// TIA Portal project "FBMECaSYSTEM_COUNTER" (V17)

(* hardware
DEVICE "HMI_1"  KTP900 Basic PN
   slot 0: "HMI_1"  KTP900 Basic PN  6AV2 123-2JB03-0AX0  17.0.0.0
   slot 1: "HMI_RT_1"  KTP900 Basic PN  6AV2 123-2JB03-0AX0  17.0.0.0
   slot 5: "HMI_1.IE_CP_1"  PROFINET Interface  17.0.0.0
      slot 1: "PROFINET Interface_1"  PROFINET Interface
         slot 1: "Port_1"  Port
DEVICE "S7-1200 station_1"  S7-1200 Station
   slot 0: "Rack_0"  S7-1200 Rack  Rack  V1.0
   slot 1: "PLC_1"  CPU 1214C AC/DC/Rly  6ES7 214-1BG40-0XB0  V4.5
*)

// ===== PLC "PLC_1"  CPU 1214C AC/DC/Rly =====

VAR_GLOBAL   // PLC tag table "Default tag table"
   "NbPersonneEntree" AT %IW10 : Int;
   "NbPersonneSortie" AT %IW14 : Int;
   "EntrerValider" AT %I20.0 : Bool;
   "SortieValider" AT %I20.1 : Bool;
   "FrontEntrerValider" AT %I20.2 : Bool;
   "FrontSortieValider" AT %I20.3 : Bool;
   "NbPersonnneInSide" AT %IW12 : Int;
   "NbPersonneTotalAutorise" AT %IW16 : Int;
   "NbPeronneRestant" AT %IW18 : Int;
   "EntreePMRValider" AT %I20.4 : Bool;
   "SortiePMRValider" AT %I20.5 : Bool;
   "NbPMR" AT %IW22 : Int;
   "FontPMRENtree" AT %I20.6 : Bool;
   "FrontPMRSortie" AT %I20.7 : Bool;
   "SitePleinQuatreVingtPC" AT %I21.0 : Bool;
   "SitePleinCentPC" AT %I21.1 : Bool;
   "FOIS80" AT %IW24 : Int;
   "DIVISER100" AT %IW26 : Int;
   "EtatRempliSite" AT %IW28 : Int;
   "Tag_1" AT %I21.2 : Bool;
   "Tag_2" AT %I21.3 : Bool;
   "Tag_3" AT %I21.4 : Bool;
   "Tag_4" AT %I21.5 : Bool;
END_VAR

ORGANIZATION_BLOCK "Main"   // OB1, LAD, ProgramCycle
TITLE = "Main Program Sweep (Cycle)"
{ S7_Optimized_Access := 'TRUE' }
VERSION : 0.1
   VAR_INPUT
      Initial_Call : Bool;   // Initial call of this OB
      Remanence : Bool;   // =True, if remanent data are available
   END_VAR
   VAR_TEMP   // added for the SCL form of the ladder/FBD networks
      _w1 : Bool;
      _w2 : Bool;
   END_VAR
BEGIN

REGION Network 1: Personne untaire entree
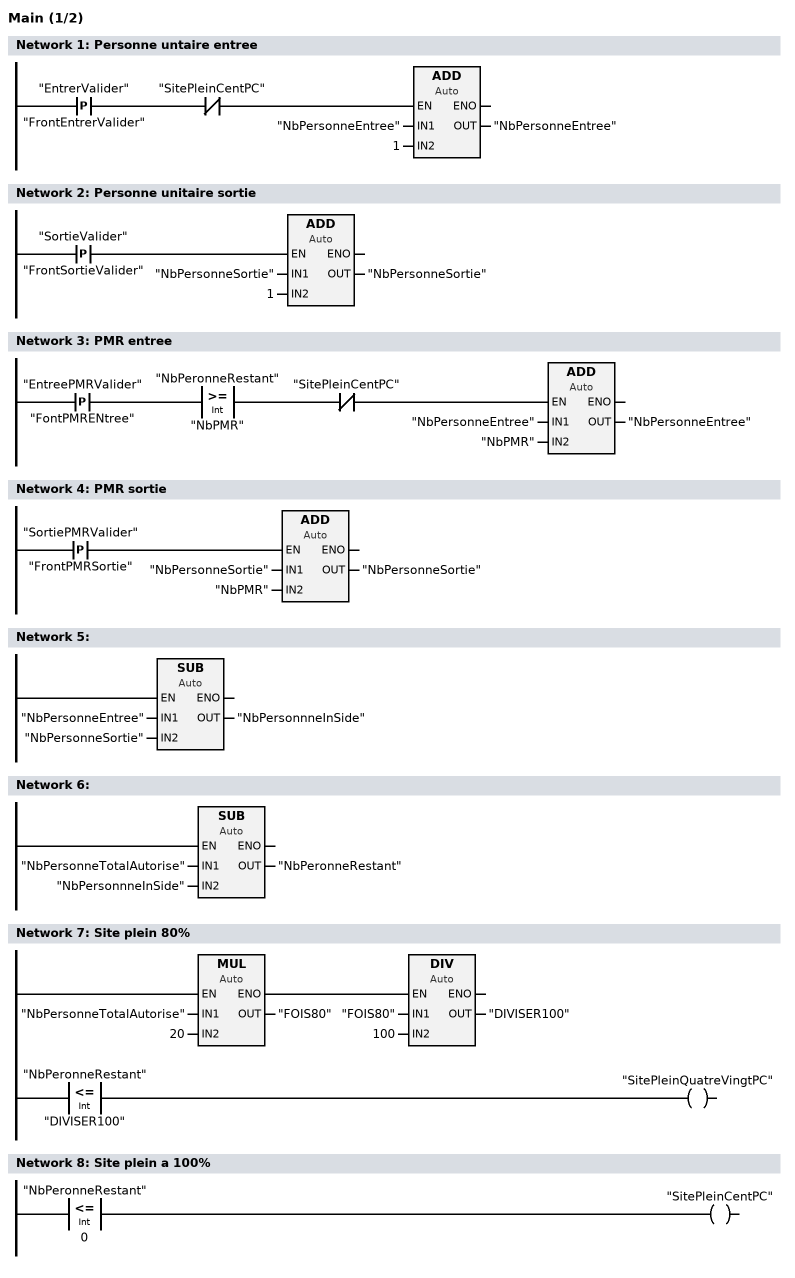
   RUNG wire#powerrail
      P_Contact(operand := "EntrerValider", bit := "FrontEntrerValider")
      I_Contact( "SitePleinCentPC" )
      Add(in1 := "NbPersonneEntree", in2 := 1, out => "NbPersonneEntree")
   END_RUNG
   // the same network as SCL:
   #_w1 := "EntrerValider" AND NOT "FrontEntrerValider";   // rising edge of "EntrerValider"
   "FrontEntrerValider" := "EntrerValider";
   IF #_w1 AND NOT "SitePleinCentPC" THEN "NbPersonneEntree" := "NbPersonneEntree" + 1; END_IF;
END_REGION

REGION Network 2: Personne unitaire sortie
   RUNG wire#powerrail
      P_Contact(operand := "SortieValider", bit := "FrontSortieValider")
      Add(in1 := "NbPersonneSortie", in2 := 1, out => "NbPersonneSortie")
   END_RUNG
   // the same network as SCL:
   #_w1 := "SortieValider" AND NOT "FrontSortieValider";   // rising edge of "SortieValider"
   "FrontSortieValider" := "SortieValider";
   IF #_w1 THEN "NbPersonneSortie" := "NbPersonneSortie" + 1; END_IF;
END_REGION

REGION Network 3: PMR entree
   RUNG wire#powerrail
      P_Contact(operand := "EntreePMRValider", bit := "FontPMRENtree")
      { S7_Templates := "SrcType := Int" } GE_Contact(in1 := "NbPeronneRestant", in2 := "NbPMR")
      I_Contact( "SitePleinCentPC" )
      Add(in1 := "NbPersonneEntree", in2 := "NbPMR", out => "NbPersonneEntree")
   END_RUNG
   // the same network as SCL:
   #_w1 := "EntreePMRValider" AND NOT "FontPMRENtree";   // rising edge of "EntreePMRValider"
   "FontPMRENtree" := "EntreePMRValider";
   IF #_w1 AND ("NbPeronneRestant" >= "NbPMR") AND NOT "SitePleinCentPC" THEN
       "NbPersonneEntree" := "NbPersonneEntree" + "NbPMR";
   END_IF;
END_REGION

REGION Network 4: PMR sortie
   RUNG wire#powerrail
      P_Contact(operand := "SortiePMRValider", bit := "FrontPMRSortie")
      Add(in1 := "NbPersonneSortie", in2 := "NbPMR", out => "NbPersonneSortie")
   END_RUNG
   // the same network as SCL:
   #_w1 := "SortiePMRValider" AND NOT "FrontPMRSortie";   // rising edge of "SortiePMRValider"
   "FrontPMRSortie" := "SortiePMRValider";
   IF #_w1 THEN "NbPersonneSortie" := "NbPersonneSortie" + "NbPMR"; END_IF;
END_REGION

REGION Network 5
   RUNG wire#powerrail
      Sub(in1 := "NbPersonneEntree", in2 := "NbPersonneSortie", out => "NbPersonnneInSide")
   END_RUNG
   // the same network as SCL:
   "NbPersonnneInSide" := "NbPersonneEntree" - "NbPersonneSortie";
END_REGION

REGION Network 6
   RUNG wire#powerrail
      Sub(in1 := "NbPersonneTotalAutorise", in2 := "NbPersonnneInSide", out => "NbPeronneRestant")
   END_RUNG
   // the same network as SCL:
   "NbPeronneRestant" := "NbPersonneTotalAutorise" - "NbPersonnneInSide";
END_REGION

REGION Network 7: Site plein 80%
   RUNG wire#powerrail
      Mul(in1 := "NbPersonneTotalAutorise", in2 := 20, out => "FOIS80")
      Div(in1 := "FOIS80", in2 := 100, out => "DIVISER100")
   END_RUNG
   RUNG wire#powerrail
      { S7_Templates := "SrcType := Int" } LE_Contact(in1 := "NbPeronneRestant", in2 := "DIVISER100")
      Coil( "SitePleinQuatreVingtPC" )
   END_RUNG
   // the same network as SCL:
   "FOIS80" := "NbPersonneTotalAutorise" * 20;
   "DIVISER100" := "FOIS80" / 100;
   "SitePleinQuatreVingtPC" := "NbPeronneRestant" <= "DIVISER100";
END_REGION

REGION Network 8: Site plein a 100%
   RUNG wire#powerrail
      { S7_Templates := "SrcType := Int" } LE_Contact(in1 := "NbPeronneRestant", in2 := 0)
      Coil( "SitePleinCentPC" )
   END_RUNG
   // the same network as SCL:
   "SitePleinCentPC" := "NbPeronneRestant" <= 0;
END_REGION

REGION Network 9
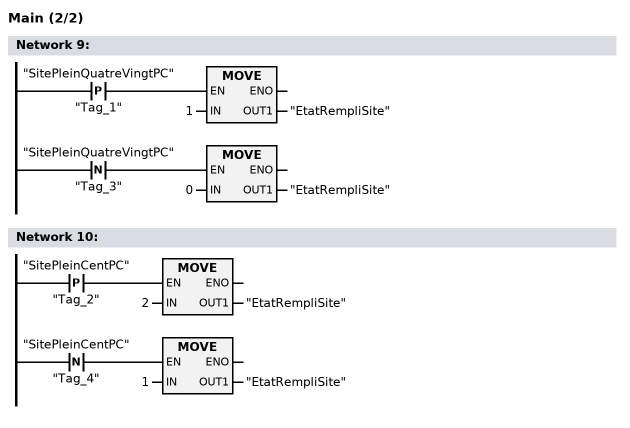
   RUNG wire#powerrail
      P_Contact(operand := "SitePleinQuatreVingtPC", bit := "Tag_1")
      Move(in := 1, out1 => "EtatRempliSite")
   END_RUNG
   RUNG wire#powerrail
      N_Contact(operand := "SitePleinQuatreVingtPC", bit := "Tag_3")
      Move(in := 0, out1 => "EtatRempliSite")
   END_RUNG
   // the same network as SCL:
   #_w1 := "SitePleinQuatreVingtPC" AND NOT "Tag_1";   // rising edge of "SitePleinQuatreVingtPC"
   "Tag_1" := "SitePleinQuatreVingtPC";
   IF #_w1 THEN "EtatRempliSite" := 1; END_IF;
   #_w2 := NOT "SitePleinQuatreVingtPC" AND "Tag_3";   // falling edge of "SitePleinQuatreVingtPC"
   "Tag_3" := "SitePleinQuatreVingtPC";
   IF #_w2 THEN "EtatRempliSite" := 0; END_IF;
END_REGION

REGION Network 10
   RUNG wire#powerrail
      P_Contact(operand := "SitePleinCentPC", bit := "Tag_2")
      Move(in := 2, out1 => "EtatRempliSite")
   END_RUNG
   RUNG wire#powerrail
      N_Contact(operand := "SitePleinCentPC", bit := "Tag_4")
      Move(in := 1, out1 => "EtatRempliSite")
   END_RUNG
   // the same network as SCL:
   #_w1 := "SitePleinCentPC" AND NOT "Tag_2";   // rising edge of "SitePleinCentPC"
   "Tag_2" := "SitePleinCentPC";
   IF #_w1 THEN "EtatRempliSite" := 2; END_IF;
   #_w2 := NOT "SitePleinCentPC" AND "Tag_4";   // falling edge of "SitePleinCentPC"
   "Tag_4" := "SitePleinCentPC";
   IF #_w2 THEN "EtatRempliSite" := 1; END_IF;
END_REGION
END_ORGANIZATION_BLOCK

ORGANIZATION_BLOCK "Startup"   // OB100, LAD, Startup
TITLE = "Complete Restart"
{ S7_Optimized_Access := 'TRUE' }
VERSION : 0.1
   VAR_INPUT
      LostRetentive : Bool;   // True if retentive data are lost
      LostRTC : Bool;   // True if date and time are lost
   END_VAR
BEGIN

REGION Network 1
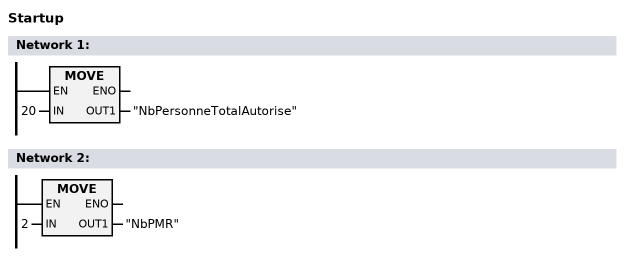
   RUNG wire#powerrail
      Move(in := 20, out1 => "NbPersonneTotalAutorise")
   END_RUNG
   // the same network as SCL:
   "NbPersonneTotalAutorise" := 20;
END_REGION

REGION Network 2
   RUNG wire#powerrail
      Move(in := 2, out1 => "NbPMR")
   END_RUNG
   // the same network as SCL:
   "NbPMR" := 2;
END_REGION
END_ORGANIZATION_BLOCK

(* ===== HMI "HMI_RT_1" =====
system functions are stored by id; their names below are inferred from use
connection "HMI_Connection_1": ETHERNET, SMART_S7_1200_OMS

HMI tags "Default tag table"
   "Tag_ScreenNumber" : UInt, internal
   "NbPersonneEntree" : Int = PLC NbPersonneEntree AT %IW10, 1 s
   "NbPersonneSortie" : Int = PLC NbPersonneSortie AT %IW14, 1 s
   "EntrerValider" : Bool = PLC EntrerValider AT %I20.0, 1 s
   "SortieValider" : Bool = PLC SortieValider AT %I20.1, 1 s
   "NbPersonnneInSide" : Int = PLC NbPersonnneInSide AT %IW12, 1 s
   "NbPersonneTotalAutorise" : Int = PLC NbPersonneTotalAutorise AT %IW16, 1 s
   "NbPeronneRestant" : Int = PLC NbPeronneRestant AT %IW18, 1 s
   "EntreePMRValider" : Bool = PLC EntreePMRValider AT %I20.4, 1 s
   "SortiePMRValider" : Bool = PLC SortiePMRValider AT %I20.5, 1 s
   "NbPMR" : Int = PLC NbPMR AT %IW22, 1 s
   "SitePleinQuatreVingtPC" : Bool = PLC SitePleinQuatreVingtPC AT %I21.0, 1 s
   "SitePleinCentPC" : Bool = PLC SitePleinCentPC AT %I21.1, 1 s
   "EtatRempliSite" : Int = PLC EtatRempliSite AT %IW28, 1 s

Template "Template_1" 800x480
   Button "Exit" at 722,440 size 55x39; TextOff 'Exit'; PictureOff "ExitRuntime_KTP900_Basic_PN_TR"; PictureOn "ExitRuntime_KTP900_Basic_PN_TR"
      on Release: StopRuntime(0)
   DateTimeField "HmiScreenItemData" at 686,35 size 105x20
   DateTimeField "HmiScreenItemData_1" at 682,7 size 105x20
   GraphicView "Template_Graphic view_1" at 28,7 size 217x65; Picture "fbmeca"

screen "Vue Princiale" 800x480, template "Template_1"
   on GenerateScreen: SetTag("Tag_ScreenNumber", 1)
   Button "Button_1" at 6,79 size 166x32; TextOff 'Entree d'une personne'
      on Press: function_b14e0dd5("EntrerValider", 0)
   Button "Button_2" at 639,79 size 161x33; TextOff 'Sortie d'une personne'
      on Press: function_b14e0dd5("SortieValider", 0)
   IOField "I/O field_3" at 296,194 size 186x92; FormatPattern 999
      ProcessValue <- "NbPersonnneInSide"
      Appearance <- "SitePleinQuatreVingtPC"
   TextField "Text field_1" at 195,145 size 409x37; Text 'Personnes à l'interieur du site'
   Button "Button_3" at 6,119 size 161x29; TextOff 'Enttrée PMR'
      on Press: function_b14e0dd5("EntreePMRValider", 0)
   Button "Button_4" at 639,116 size 161x29; TextOff 'Sortie PMR'
      on Press: function_b14e0dd5("SortiePMRValider", 0)
   IOField "I/O field_1" at 330,348 size 126x58; FormatPattern 999
      ProcessValue <- "NbPersonneTotalAutorise"
   TextField "Text field_2" at 201,321 size 376x29; Text 'Nombre Max de Personnes autorisé'
   TextField "Text field_3" at 320,449 size 33x20; Text 'Text'
      Visibility <- "EtatRempliSite"
   Softkey "Softkey_F1" at 0,0 size 0x0
      on KeyDown: ActivateScreen("Vue Parametrage", 0)

screen "Vue Parametrage" 800x480
   TextField "Text field_1" at 3,51 size 303x29; Text 'Nombre de Peronne autorisé'
   IOField "I/O field_1" at 394,38 size 96x32; FormatPattern s99999
      ProcessValue <- "NbPersonneTotalAutorise"
   TextField "Text field_2" at 3,96 size 319x29; Text 'Nombre de Peronne avec PMR'
   IOField "I/O field_2" at 394,93 size 96x32; FormatPattern s99999
      ProcessValue <- "NbPMR"
   Softkey "Softkey_F1" at 0,0 size 0x0
      on KeyDown: ActivateScreen("Vue Princiale", 0)
*)